// TIA Portal V17 export
VAR_GLOBAL   // PLC tag table "Tags_Elevador"
   Botao_sobe_1 AT %I0.0 : Bool;   // Botão de impulso contato N.O. painel de comando no 1º pavimento
   Botao_desce_1 AT %I0.1 : Bool;   // Botão de impulso contato N.O. painel de comando no 1º pavimento
   Fim_de_curso_da_cabine_1 AT %I0.2 : Bool;   // Chave fim de curso contato N.C. posição da cabine no 1º pavimento
   Fim_de_curso_da_porta_1 AT %I0.3 : Bool;   // Chave fim de curso contato N.O. posição da porta no 1º pavimento
   Botao_sobe_2 AT %I0.4 : Bool;   // Botão de impulso contato N.O. painel de comando no 2º pavimento
   Botao_desce_2 AT %I0.5 : Bool;   // Botão de impulso contato N.O. painel de comando no 2º pavimento
   Fim_de_curso_da_cabine_2 AT %I0.6 : Bool;   // Chave fim de curso contato N.C. posição da cabine no 2º pavimento
   Fim_de_curso_da_porta_2 AT %I0.7 : Bool;   // Chave fim de curso contato N.O. posição da porta no 2º pavimento
   Motor_1_sobe AT %Q0.0 : Bool;   // Motor com sentido de rotação para subir a cabine (horário)
   Motor_1_desce AT %Q0.1 : Bool;   // Motor com sentido de rotação para descer a cabine (anti-horário)
   Tranca_magnetica_da_porta_1 AT %Q0.2 : Bool;   // Tranca magnética da porta do 1º pavimento
   Tranca_magnetica_da_porta_2 AT %Q0.3 : Bool;   // Tranca magnética da porta do 2º pavimento
END_VAR
